// TIA Portal V16 export
// export: Created 2025-05-24T14:07:40.1018083Z, ExportSetting WithDefaults, DisplayName Totally Integrated Automation Portal, DisplayVersion V16, DisplayName TIA Portal Version Control Interface, DisplayVersion V16, DisplayName TIA Portal Openness, DisplayVersion V16, DisplayName STEP 7 Professional, DisplayVersion V16, DisplayName STEP 7 Safety, DisplayVersion V16, DisplayName WinCC Advanced, DisplayVersion V16
FUNCTION_BLOCK "Alarm_Axis_Position_Function"   // FB3, FBD
TITLE = Alarm Axis not in Position
VERSION : 0.1
// stored: AutoNumber true, IsIECCheckEnabled false, UDAEnableTagReadback false
   VAR_INPUT
      "Axis FWD command" : Bool;
      "Axis Feedback (Sensor) signal" : Bool;
      "Axis Encoder Singal" : Real;
      "Axis Command Position" : Real;
      "Sensor Controlled (HIGH) - Position Controlled (LOW)" : Bool;
      "CheckTime Setting" : Time := T#5S;
   END_VAR
   VAR_OUTPUT
      "Alarm BOOL" : Bool;
      "Alarm WORD" : Bool;
   END_VAR
   VAR_TEMP
      "Axis Feedback Internal" : Bool;
      "Axis Encoder On Position" : Bool;
      "Axis Sensor On Position" : Bool;
      "Axis Measuring Mode" : Bool;
   END_VAR
BEGIN

REGION Network 1: When axis is spinning start timer
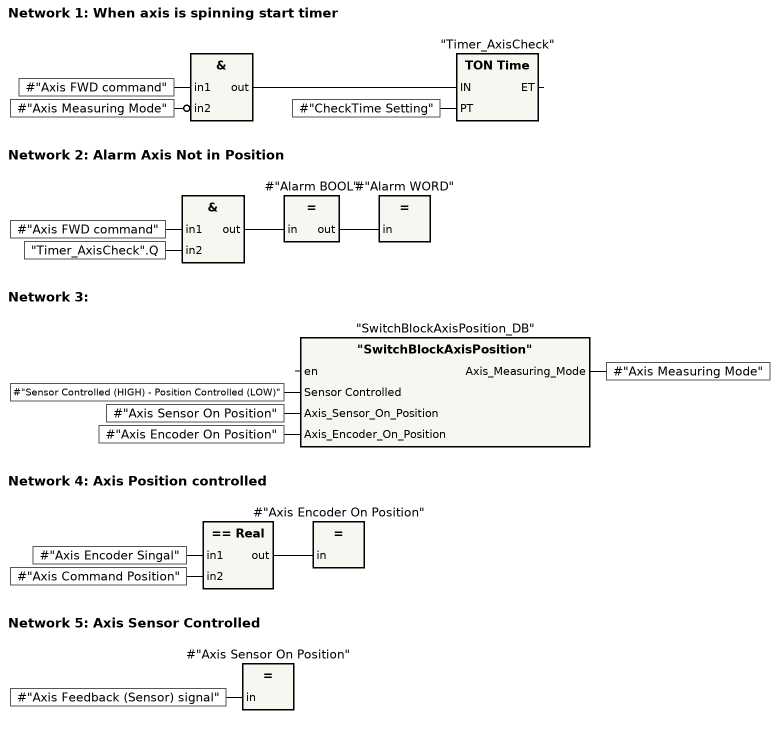
   "Timer_AxisCheck".TON(IN := #"Axis FWD command" AND NOT #"Axis Measuring Mode", PT := #"CheckTime Setting");
END_REGION

REGION Network 2: Alarm Axis Not in Position
   #"Alarm BOOL" := #"Axis FWD command" AND "Timer_AxisCheck".Q;
   #"Alarm WORD" := #"Alarm BOOL";
END_REGION

REGION Network 3
   "SwitchBlockAxisPosition_DB"("Sensor Controlled" := #"Sensor Controlled (HIGH) - Position Controlled (LOW)",   // "SwitchBlockAxisPosition"
                           Axis_Sensor_On_Position := #"Axis Sensor On Position",
                           Axis_Encoder_On_Position := #"Axis Encoder On Position",
                           Axis_Measuring_Mode => #"Axis Measuring Mode");
END_REGION

REGION Network 4: Axis Position controlled
   #"Axis Encoder On Position" := #"Axis Encoder Singal" = #"Axis Command Position";
END_REGION

REGION Network 5: Axis Sensor Controlled
   #"Axis Sensor On Position" := #"Axis Feedback (Sensor) signal";
END_REGION
END_FUNCTION_BLOCK
